{attribute 'linkalways'} 
{attribute 'no_explicit_call' := 'This FB is a CLASS and must be accessed using methods or properties'}
{attribute 'enable_dynamic_creation'}
FUNCTION_BLOCK _MyStruct EXTENDS StructuredDatatypeBase
VAR
	localData : MyStruct;
	activeData : REFERENCE TO MyStruct REF= localData;
	_myBit : _BIT;
END_VAR

PROPERTY PUBLIC Address : PVOID
GET
Address := ADR(activeData);
END_GET
END_PROPERTY

METHOD PUBLIC ClearReference
VAR_INPUT
END_VAR
activeData REF= localData;
SetMemberReference();
END_METHOD

METHOD PUBLIC Clone : I_Datatype
VAR
    pClone : POINTER TO _MyStruct;
END_VAR
pClone := __NEW(_MyStruct());
pClone^.Value := Value;
Clone := pClone^;
END_METHOD

METHOD FB_init : BOOL
VAR_INPUT
	bInitRetains : BOOL; // if TRUE, the retain variables are initialized (warm start / cold start)
	bInCopyCode : BOOL;  // if TRUE, the instance afterwards gets moved into the copy code (online change)
END_VAR
SetMemberReference();
AddMember('MyBit',_myBit);
END_METHOD

PROPERTY PUBLIC Identifier : T_MAXSTRING
GET
Identifier := 'MyStruct';
END_GET
END_PROPERTY

METHOD PUBLIC MakeReferenceTo
VAR_INPUT
	ReferenceTarget : REFERENCE TO MyStruct;
END_VAR
activeData REF= ReferenceTarget;
SetMemberReference();
END_METHOD

PROPERTY PUBLIC MyBit : Reference to _BIT
GET
MyBit REF= _myBit;
END_GET
END_PROPERTY

METHOD PROTECTED SetMemberReference
VAR_STAT
	// this variable is used for BITADR as this function failes if used on a local variable.
	structure : MyStruct;
END_VAR
_myBit.MakeReferenceTo(THIS^, GetByteOffset(localData, localData.MyBit), BITADR(structure.MyBit));
END_METHOD

PROPERTY PUBLIC Size : UDINT
GET
Size := SIZEOF(activeData);
END_GET
END_PROPERTY

METHOD TryMakeReferenceTo : BOOL
VAR_INPUT
	Target : I_Datatype;
END_VAR
VAR
	pTargetData : POINTER TO MyStruct;
END_VAR
IF NOT IsEquivalentTo(Target) THEN
	RETURN;
END_IF

pTargetData := Target.Address;
activeData REF= pTargetData^;
SetMemberReference();
TryMakeReferenceTo := TRUE;
END_METHOD

PROPERTY PUBLIC Value : REFERENCE TO MyStruct
GET
Value REF= activeData;
END_GET
END_PROPERTY

END_FUNCTION_BLOCK

(* stored: Version 1.1.0.1, ProductVersion 3.1.4024.13
   POU _MyStruct: Id {c95335ad-c5c5-4ca4-9b81-670617e863ba}, SpecialFunc None
   Folder Constructor: Id {eaaac4e9-8a4a-4550-83d9-082c7c28fb26}
   Folder Protected: Id {49958b28-32ac-4d79-9360-30bbd7bb0fe8}
   Property Address: Id {ad48cdfe-cdef-465c-b5f0-8f67d138a17f}
   Get Get: Id {df9eaff3-1cb4-4c2b-b948-d98c5c81130d}
   Method ClearReference: Id {083d7841-7ead-4963-8bb6-6730125c51c9}
   Method Clone: Id {c9244f1d-803c-483d-9d81-ccd6e1612835}
   Method FB_init: Id {e810e1b0-d92c-4f38-95ae-3f0480fbf27d}
   Property Identifier: Id {25ebb523-d078-4916-ba0a-ee8e880f70c4}
   Get Get: Id {90a80ab6-6cdb-4a13-a2d5-6ee207079295}
   Method MakeReferenceTo: Id {fc4d1ba3-334d-4f71-aaf5-3c3d0ddc3ddf}
   Property MyBit: Id {c69fdd62-05e2-464d-bd70-a88f3181d120}
   Get Get: Id {ff3cb494-b5d4-46fb-98a9-83a13076991b}
   Method SetMemberReference: Id {b2d29e80-536a-46f0-b53a-ea8e76601be6}
   Property Size: Id {74d051e4-7162-4209-9df9-958ebf74e194}
   Get Get: Id {b159b6d0-e49b-48d4-a9bf-cee0f3fbf4a3}
   Method TryMakeReferenceTo: Id {87b54037-7b95-4e7e-89a5-f85475e6850e}
   Property Value: Id {78169baa-8f82-4435-9209-e699506fed47}
   Get Get: Id {7e7d3f34-1164-4ad4-b630-fc4c7717e0ce} *)
